PROGRAM MAIN
VAR
	fbAPS_Prog:FB_APS_Prog;
END_VAR

fbAPS_Prog();

END_PROGRAM

(* stored: Version 1.1.0.1, ProductVersion 3.1.4024.12
   POU MAIN: Id {0a9ebfbe-586c-4bb2-b52a-ab34082263a2}, SpecialFunc None *)
